// TIA Portal V20 export
TYPE "DigitalOutput_DT"
   STRUCT
      SWStatus : Bool;   // Software status use in PLC code
      HWStatus : Bool;   // Hardware status directly set to physical output
   END_STRUCT;
END_TYPE
